PROGRAM MAIN
VAR
	fHysteresis: REAL := 1;		//Hysteresis value
	rUpperLimit: REAL;		 	//Temperature set value added with Hysteresis
	rLowerLimit: REAL;		 	//Temperature set value subtracted with Hysteresis
END_VAR

rUpperLimit := GVL_Var.fTempSet + fHysteresis;
rLowerLimit := GVL_Var.fTempSet - fHysteresis;

// Logic to switch ON the compressor when it exceeds the UpperLimit
// and compressor switched OFF when it is below the lowerLimit
IF GVL_Var.fTempActual > rUpperLimit THEN
	GVL_Var.bCompressor := TRUE;
ELSIF GVL_Var.fTempActual < rLowerLimit THEN
	GVL_Var.bCompressor := FALSE; 
END_IF

//Calling Signal1 Program
Signal1();

END_PROGRAM

(* stored: Version 1.1.0.1, ProductVersion 3.1.4024.4
   POU MAIN: Id {99dfa53b-5419-4e73-b545-8a9f1a8f4f63}, SpecialFunc None *)
